// TwinCAT 3 PLC project festoArmPlc
// ProgramVersion: 3.1.4022.1
// libraries:
//   Tc2_MC2, * (Beckhoff Automation GmbH)
//   Tc2_SerialCom, * (Beckhoff Automation GmbH)
//   Tc2_Standard, * (Beckhoff Automation GmbH)
//   Tc2_System, * (Beckhoff Automation GmbH)
//   Tc3_Module, * (Beckhoff Automation GmbH)
// project tree:
//   / PlcTask.TcTTO
//   POUs/ MAIN.TcPOU, SerialRecieve.TcPOU
// real-time tasks:
//   TASK cpp: cycle T#10ms, priority 1, ADS port 350
//   TASK PlcTask: cycle T#10ms, priority 20, ADS port 351
// motion (NC):
//   TASK NC-Task 1 SAF: cycle T#2ms, priority 4, ADS port 501
//   TASK NC-Task 1 SVB: cycle T#10ms, priority 8, ADS port 511
//   AXIS AxisShoulderLevelShift (id 1)
//     Velo: SlowManual=0.5, FastManual=2, Maximum=8
//     OtherSettings: AllowMotionCmdToSlave=true
//     encoder EncType=19
//       EncPara: ScaleFactorNumerator=360, ScaleFactorDenominator=942080, MaxCount=#xffffffff
//     drive DrvType=16
//       DrvPara: MaxCount=#xffffffff
//         Analog: VeloReferenz=7
//         TimeComp: TaskDelayCycles=1
//     controller CtrType=1
//       CtrPara: PriorControlFactor=1
//         Observer: BandWidth=20
//   AXIS AxisShoulderRotate (id 2)
//     Velo: SlowManual=0.5, FastManual=2, Maximum=8
//     OtherSettings: AllowMotionCmdToSlave=true
//     encoder EncType=19
//       EncPara: ScaleFactorNumerator=360, ScaleFactorDenominator=942080, MaxCount=#xffffffff
//     drive DrvType=16
//       DrvPara: MaxCount=#xffffffff
//         Analog: VeloReferenz=7
//         TimeComp: TaskDelayCycles=1
//     controller CtrType=1
//       CtrPara: PriorControlFactor=1
//         Observer: BandWidth=20
// I/O:
//   DEVICE Device 1 (EtherCAT), AmsNetId 5.39.221.128.2.1
//     Term 1 (EK1200) [EK1200-5000 EtherCAT Power supply (2A E-Bus)]
//       Term 2 (EL6001) [EL6001 Interface (RS232)]
//       Term 7 (EK1122) [EK1122 2 port EtherCAT junction]
//         Drive 3 (Elmo Drive) [Gold EtherCAT GCON Drive Rev:0x000103F6]
//         Drive 5 (Elmo Drive) [Gold EtherCAT GCON Drive Rev:0x000103F6]
//   DEVICE Device 4 (EtherCAT), AmsNetId 5.39.221.128.5.1
//     Box 4 (CPX-FB37) [CPX-FB37 Fieldbus module]
//       modules: Module 1 (FB37-RIO), elbow2, elbow1, Module 4 (VPPM Display 10 bar [1AI/1AO]), wrist, Module 6 (VPPM Display 10 bar [1AI/1AO]), Module 7 (VPPM Display 10 bar [1AI/1AO]), Module 8 (VPPM Display 10 bar [1AI/1AO]), Module 9 (VPPM Display 10 bar [1AI/1AO])
// variable links:
//   NC-Task 1 SAF/Axes/AxisShoulderLevelShift <-> Device 1 (EtherCAT)/Term 1 (EK1200)/Term 7 (EK1122)/Drive 3 (Elmo Drive)
//     Drive/Inputs/In/nDcOutputTime <-> InfoData/DcOutputShift
//     Drive/Inputs/In/nState1 <-> Inputs/Status word
//     Drive/Inputs/In/nState2 <-> Inputs/Status word @bit 8
//     Drive/Inputs/In/nState4 @bit 1 <-> WcState/InputToggle
//     Drive/Inputs/In/nState4 <-> WcState/WcState
//     Drive/Outputs/Out/nCtrl1 <-> Outputs/Control word
//     Drive/Outputs/Out/nCtrl2 <-> Outputs/Control word @bit 8
//     Drive/Outputs/Out/nDataOut1 <-> Outputs/Target Position
//     Enc/Inputs/In/nDataIn1 <-> Inputs/Position actual value
//     Enc/Inputs/In/nDcInputTime <-> InfoData/DcInputShift
//     Enc/Inputs/In/nState4 @bit 1 <-> WcState/InputToggle
//     Enc/Inputs/In/nState4 <-> WcState/WcState
//   NC-Task 1 SAF/Axes/AxisShoulderRotate <-> Device 1 (EtherCAT)/Term 1 (EK1200)/Term 7 (EK1122)/Drive 5 (Elmo Drive)
//     Drive/Inputs/In/nDcOutputTime <-> InfoData/DcOutputShift
//     Drive/Inputs/In/nState1 <-> Inputs/Status word
//     Drive/Inputs/In/nState2 <-> Inputs/Status word @bit 8
//     Drive/Inputs/In/nState4 @bit 1 <-> WcState/InputToggle
//     Drive/Inputs/In/nState4 <-> WcState/WcState
//     Drive/Outputs/Out/nCtrl1 <-> Outputs/Control word
//     Drive/Outputs/Out/nCtrl2 <-> Outputs/Control word @bit 8
//     Drive/Outputs/Out/nDataOut1 <-> Outputs/Target Position
//     Enc/Inputs/In/nDataIn1 <-> Inputs/Position actual value
//     Enc/Inputs/In/nDcInputTime <-> InfoData/DcInputShift
//     Enc/Inputs/In/nState4 @bit 1 <-> WcState/InputToggle
//     Enc/Inputs/In/nState4 <-> WcState/WcState
//   festoArmPlc/festoArmPlc Instance <-> Device 1 (EtherCAT)/Term 1 (EK1200)/Term 2 (EL6001)
//     PlcTask Inputs/SerialRecieve.EL6_22Bin_PC1/D <-> COM Inputs/Data In 0
//     PlcTask Inputs/SerialRecieve.EL6_22Bin_PC1/D @bit {8..168 step 8} <-> COM Inputs/Data In {1..21}  (21 links)
//     PlcTask Inputs/SerialRecieve.EL6_22Bin_PC1/Status <-> COM Inputs/Status
//     PlcTask Outputs/SerialRecieve.EL6_22Bout_PC1/Ctrl <-> COM Outputs/Ctrl
//     PlcTask Outputs/SerialRecieve.EL6_22Bout_PC1/D <-> COM Outputs/Data Out 0
//     PlcTask Outputs/SerialRecieve.EL6_22Bout_PC1/D @bit {8..168 step 8} <-> COM Outputs/Data Out {1..21}  (21 links)
//   festoArmPlc/festoArmPlc Instance <-> Device 4 (EtherCAT)/Box 4 (CPX-FB37)
//     PlcTask Outputs/MAIN.elbow1 <-> elbow1/Outputs/elbow1Output
//     PlcTask Outputs/MAIN.elbow2 <-> elbow2/Outputs/elbow2Output
//     PlcTask Outputs/MAIN.wrist <-> wrist/Outputs/wristOutput
//   festoArmPlc/festoArmPlc Instance <-> NC-Task 1 SAF/Axes/AxisShoulderLevelShift
//     PlcTask Inputs/MAIN.AxisLevelShift.NcToPlc <-> Outputs/ToPlc
//     PlcTask Outputs/MAIN.AxisLevelShift.PlcToNc <-> Inputs/FromPlc
//   festoArmPlc/festoArmPlc Instance <-> NC-Task 1 SAF/Axes/AxisShoulderRotate
//     PlcTask Inputs/MAIN.AxisRotate.NcToPlc <-> Outputs/ToPlc
//     PlcTask Outputs/MAIN.AxisRotate.PlcToNc <-> Inputs/FromPlc

CONFIGURATION festoArmPlc
    RESOURCE PLC ON TwinCAT3
        TASK PlcTask(INTERVAL := T#10ms, PRIORITY := 20);
        PROGRAM MAIN WITH PlcTask : MAIN;
        PROGRAM SerialRecieve WITH PlcTask : SerialRecieve;
    END_RESOURCE
END_CONFIGURATION

// ---- POUs/MAIN.TcPOU
PROGRAM MAIN
VAR
	elbow1, elbow2 AT%Q* : INT;
	BILI1, BILI2: LREAL;
	wrist AT%Q* : INT;
	wrist_real : LREAL;
	
	//肩关节水平移动自由度变量
	AxisLevelShift: AXIS_REF;											//运动轴
	MC_PowerLevelShift: MC_Power;										//电源模块
	MC_MoveAbsoluteLevelShift: MC_MoveAbsolute;							//绝对运动模块
	
	//肩关节旋转移动自由度变量
	AxisRotate: AXIS_REF;												//运动轴
	MC_PowerRotate: MC_Power;											//电源模块
	MC_MoveAbsoluteRotate: MC_MoveAbsolute;								//绝对运动模块
	
	//肩关节初始化完成标志量
	ShoulderInitStart AT%I* : BOOL := TRUE;							//肩关节初始化启动
	ShoulderInitFinish AT%Q*: BOOL := FALSE;
	
	//PLC时间
	Timer AT%Q*: LREAL := 0;											//时间 
	InitStatusLevelShift: INT;
	ErrorTime: LREAL;
	InitFinishLevelShift: BOOL;
	ErrorCode: INT;
	InitStatusRotate: INT;
	InitFinishRotate: BOOL;
	MC_MoveAbsolute1: INT;
	startTimer: LREAL;
	sTime: LREAL;
	holdTime: LREAL;
END_VAR

MC_PowerLevelShift(
	Axis:= AxisLevelShift,
	Enable_Positive:= TRUE,
	Enable_Negative:= TRUE, );
	
MC_MoveAbsoluteLevelShift(
	Axis:= AxisLevelShift, );
	
MC_PowerRotate(
	Axis:= AxisRotate,
	Enable_Positive:= TRUE,
	Enable_Negative:= TRUE, );
	
MC_MoveAbsoluteRotate(
	Axis:= AxisRotate, );
		
IF ShoulderInitFinish = FALSE THEN
	//肩关节初始化
	
	//平移自由度
	
	CASE InitStatusLevelShift OF
		0://等待初始化命令
			IF ShoulderInitStart THEN
				InitStatusLevelShift := 1;
			END_IF
		1://init 初始化
			MC_PowerLevelShift.Enable := FALSE;
			MC_MoveAbsoluteLevelShift.Execute := FALSE;
			InitStatusLevelShift := 2;
		2://power 使能
			MC_PowerLevelShift.Enable := TRUE;
			IF MC_PowerLevelShift.Status THEN
				InitStatusLevelShift := 3;
			END_IF
			IF AxisLevelShift.Status.Error THEN
				//ErrorTime := Timer;
				InitStatusLevelShift := 5;
			END_IF
		3://move 移动到初始位置
			MC_MoveAbsoluteLevelShift.Position := 0;
			MC_MoveAbsoluteLevelShift.Velocity := 3;
			MC_MoveAbsoluteLevelShift.Execute := TRUE;
			IF MC_MoveAbsoluteLevelShift.Done THEN
				MC_MoveAbsoluteLevelShift.Execute := FALSE;
				InitStatusLevelShift := 4;
			END_IF
		4://finishInit 初始化完成
			InitFinishLevelShift := TRUE;
		5://error
			ErrorCode := 1000;
	END_CASE
	
	
	//旋转自由度
	
	CASE InitStatusRotate OF
		0://等待初始化命令
			IF ShoulderInitStart THEN
				InitStatusRotate := 1;
			END_IF
		1://init 初始化
			MC_PowerRotate.Enable := FALSE;
			MC_MoveAbsoluteRotate.Execute := FALSE;
			InitStatusRotate := 2;
		2://power 使能
			MC_PowerRotate.Enable := TRUE;
			IF MC_PowerRotate.Status THEN
				InitStatusRotate := 3;
			END_IF
			IF AxisLevelShift.Status.Error THEN
				//ErrorTime := Timer;
				InitStatusRotate := 5;
			END_IF
		3://move 移动到初始位置
			MC_MoveAbsoluteRotate.Position := 0;
			MC_MoveAbsoluteRotate.Velocity := 3;
			MC_MoveAbsoluteRotate.Execute := TRUE;
			IF MC_MoveAbsoluteRotate.Done THEN
				MC_MoveAbsoluteRotate.Execute := FALSE;
				InitStatusRotate := 4;
			END_IF
		4://finishInit 初始化完成
			InitFinishRotate := TRUE;
		5://error
			ErrorCode := 1100;
	END_CASE
			
	IF InitFinishLevelShift AND InitFinishRotate THEN
		ShoulderInitFinish := TRUE;
	END_IF
END_IF

IF ShoulderInitFinish = TRUE THEN
	Timer := Timer + 0.01;
	
	IF Timer < 10 THEN	//电机移动
		MC_MoveAbsoluteLevelShift.Position := 25;
		MC_MoveAbsoluteLevelShift.Velocity := 4;
		MC_MoveAbsoluteLevelShift.Execute := TRUE;
	END_IF
	
	IF Timer > 10 AND Timer < 20 THEN //初始化
		BILI1 := (Timer - 10) / 10.0 * 2.7;
		BILI2 := 0;
	END_IF
	
	IF Timer > 20 AND Timer < 30 THEN //肘关节动
		BILI1 := 2.5;
		BILI2 := (Timer - 20) / 10.0 * 3.0;
	END_IF
	
	IF Timer > 30 AND Timer < 40 THEN //腕关节动
		wrist_real := (Timer - 30) / 10.0 * 6.0;
	END_IF
	
	IF Timer > 50 AND Timer < 60 THEN //肘关节放气
		//BILI1 := (60 - Timer) / 10.0 * 2.7;
		BILI2 := (60 - Timer) / 10.0 * 3.0;
	END_IF
	
	IF Timer > 60 AND Timer < 70 THEN //腕关节放气
		wrist_real := (70 - Timer) / 10.0 * 6.0;
	END_IF
	
	(*IF Timer > 70 AND Timer < 80 THEN //腕关节放气
		MC_MoveAbsoluteLevelShift.Execute := FALSE;
		MC_MoveAbsoluteLevelShift.Position := 0;
		MC_MoveAbsoluteLevelShift.Velocity := 4;
		MC_MoveAbsoluteLevelShift.Execute := TRUE;
	END_IF*)
END_IF

//输出
IF BILI1 < 46 AND BILI2 < 6 THEN
	elbow1 := LREAL_TO_INT(BILI1 / 10.0 * 10000);
	elbow2 := LREAL_TO_INT(BILI2 / 10.0 * 10000);
END_IF
IF wrist_real < 7 THEN
	wrist := LREAL_TO_INT(wrist_real / 10.0 * 10000);
END_IF

END_PROGRAM

// ---- POUs/SerialRecieve.TcPOU
PROGRAM SerialRecieve
VAR
	//读取编码器角度
	EL6_22Bin_PC1	AT %I* 	: KL6inData22b;
	EL6_22Bout_PC1	AT %Q*	: KL6outData22b;
	RxBuffer1: COMBuffer;
	TxBuffer1: COMBuffer;
	JIAODU	AT %Q* : LREAL;(*单位 度*)
	JIAOSUDU: LREAL;(*单位 度*)
	JIAOJIASUDU: LREAL;(*单位 度*)
	SerialLineControlElbow:SerialLineControl;
	
	i:INT;
    AA:BYTE;
	BB:BYTE;
	RxBufferStep:INT:=0;
    AA_P:BYTE;
	BB_P:BYTE;
	JIAODU_INT:INT;
	J1: LREAL:=0;
	J2: LREAL:=0;
	J3: LREAL:=0;
	W1: LREAL:=0;
	W2: LREAL:=0;
	t_tip: LREAL:=0.01;
END_VAR

//读取编码器的数值
SerialLineControlElbow(
	Mode:= SERIALLINEMODE_KL6_22B_STANDARD, 
	pComIn:= ADR(EL6_22Bin_PC1), 
	pComOut:= ADR(EL6_22Bout_PC1), 
	SizeComIn:= UINT_TO_INT(SIZEOF(EL6_22Bin_PC1)), 
	TxBuffer:= TxBuffer1, 
	RxBuffer:= RxBuffer1);

IF RxBuffer1.Count<> 0 THEN
	FOR i:=1 TO UINT_TO_INT(RxBuffer1.Count) DO
		IF RxBufferStep=3 THEN
			BB:=RxBuffer1.Buffer[RxBuffer1.RdIdx];
			AA:=AA_P;
			RxBufferStep:=0;
		END_IF
		IF RxBufferStep=2 THEN
			AA_P:=RxBuffer1.Buffer[RxBuffer1.RdIdx];
			RxBufferStep:=3;
		END_IF
		IF RxBufferStep=1 THEN
			IF RxBuffer1.Buffer[RxBuffer1.RdIdx]=90 THEN
				RxBufferStep:=2;
			ELSE
				RxBufferStep:=0;
			END_IF
		END_IF
		IF RxBuffer1.Buffer[RxBuffer1.RdIdx]=165 THEN
			RxBufferStep:=1;
		END_IF

		RxBuffer1.RdIdx:=RxBuffer1.RdIdx+1;
		IF RxBuffer1.RdIdx>300 THEN
			RxBuffer1.RdIdx:=0;
		END_IF
	END_FOR
RxBuffer1.Count:=0;
END_IF

JIAODU_INT:=UINT_TO_INT(AA*256+BB);
JIAODU:=INT_TO_REAL(JIAODU_INT)*360.0/4096.0;
J3:=J2;
J2:=J1;
J1:=JIAODU;
JIAOSUDU:=(J1-J2)/t_tip;
W2:=W1;
W1:=JIAOSUDU;
JIAOJIASUDU:=(W1-W2)/t_tip;

END_PROGRAM
